// Mitsubishi GX Works2 project: a8   PLC: Q02/Q02H

PROGRAM MAIN
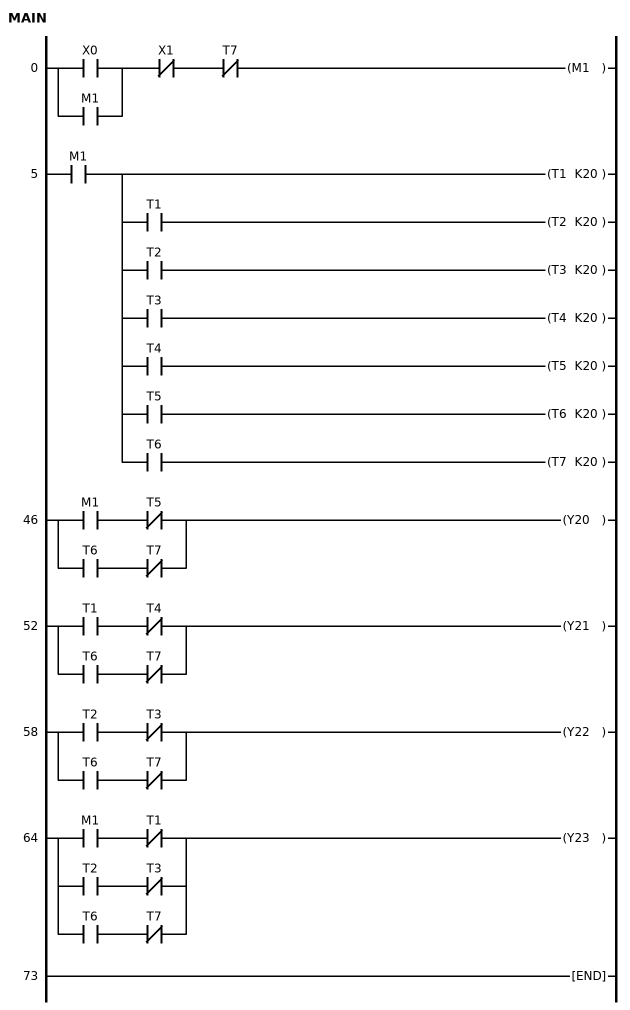
0     LD      X0
      OR      M1
      ANI     X1
      ANI     T7
      OUT     M1
5     LD      M1
      OUT     T1 K20
      MPS
      AND     T1
      OUT     T2 K20
      MRD
      AND     T2
      OUT     T3 K20
      MRD
      AND     T3
      OUT     T4 K20
      MRD
      AND     T4
      OUT     T5 K20
      MRD
      AND     T5
      OUT     T6 K20
      MPP
      AND     T6
      OUT     T7 K20
46    LD      M1
      ANI     T5
      LD      T6
      ANI     T7
      ORB
      OUT     Y20
52    LD      T1
      ANI     T4
      LD      T6
      ANI     T7
      ORB
      OUT     Y21
58    LD      T2
      ANI     T3
      LD      T6
      ANI     T7
      ORB
      OUT     Y22
64    LD      M1
      ANI     T1
      LD      T2
      ANI     T3
      ORB
      LD      T6
      ANI     T7
      ORB
      OUT     Y23
73    END
END_PROGRAM
